Staubli VAL3: start.pgx

program start()
begin
  //利用4毫秒来实现同步功能














end
